FUNCTION_BLOCK FB_DigitalOut IMPLEMENTS I_DigitalOut
VAR_INPUT
END_VAR
VAR_OUTPUT
	bOutput AT %Q* : BOOL := FALSE;
END_VAR
VAR
END_VAR

METHOD M_Off
bOutput := FALSE;
END_METHOD

METHOD M_On
bOutput := TRUE;
END_METHOD

END_FUNCTION_BLOCK

(* stored: Version 1.1.0.1, ProductVersion 3.1.0.19
   POU FB_DigitalOut: Id {3ff8d448-d7cf-462d-8b2e-ff592af894bf}
   Method M_Off: Id {f480b60d-2691-4e51-8ebe-8e6447390bbb}
   Method M_On: Id {45b5ab3a-8962-4617-89c5-df4059cd36fa} *)
